//-----------------------------------------------------------------------------------------------------
//																
//									 	Tkmatik sp z o.o.
//
//	Name					:		FB_Save
//	Author					:		AM
//	Release Date			:		12.01.2022
//	Current ver				:		v 0.1
// 	Last correction 		:		12.01.2022
// 
//	Description				:
//		Special FB for saving structures to CSV files						
//
//	Requared hardware		:
//
// 	Configuration			:
//
//
//-----------------------------------------------------------------------------------------------------

FUNCTION_BLOCK FB_RecipeVariablesSaveCSV

VAR_INPUT
	bExecute							: BOOL := FALSE;(* Rising edge starts program execution *)
	sFilePath							: T_MaxString;(* CSV destination file path and name *)
//	database							: POINTER TO STRING(255);	
	nRows          						: UDINT;                // Liczba wierszy
    nCols          						: UDINT; 
	database							: POINTER TO STRING(255);//ARRAY[0..MAX_PARAMS_VARIABLES_COUNT-1] OF STRING(255);
	
END_VAR
VAR CONSTANT
	MAX_CSV_FIELD_LENGTH				: UDINT	:= 255;	
END_VAR
VAR_IN_OUT
END_VAR

VAR
	
	sNetId			: T_AmsNetId := '';	(* TwinCAT system network address *)
	sCSVLine		: T_MaxString := '';(* Single CSV text line (row, record), we are using string as record buffer (your are able to see created fields) *)
	sCSVField		: T_MaxString := '';(* Single CSV field value (column, record field) *)
	nRow	 		: UDINT 	:= 0;(* Row number (record) *)
	nColumn			: UDINT 	:= 0;(* Column number (record field) *)
	hFile			: UINT		:= 0;(* File handle of the source file *)
	step			: DWORD 	:= 0;
	fbFileOpen		: FB_FileOpen;(* Opens file *)
	fbFileClose		: FB_FileClose;(* Closes file *)
	fbFilePuts		: FB_FilePuts;(* Writes one record (line) *)
	fbWriter		: FB_CSVMemBufferWriter;(* Helper function block used to create CSV data bytes (single record line) *)
	rtExecute		:	R_TRIG;                         //	Rtrig for start



END_VAR
VAR_OUTPUT                                                                                  
	bBusy												:	BOOL;                           //	FB is Busy
	bDone												:	BOOL;                           //	Load cycle done, DATA actual 
	bError												:	BOOL;                           //	Flag error
	nErrId												:	UDINT;                          //	Error ID

END_VAR


rtExecute(CLK:=bExecute);
IF (NOT bExecute) THEN
	bDone												:=	FALSE;
END_IF

CASE step OF
	0:	(* Wait for rising edge at bWrite variable *)
		IF rtExecute.Q THEN
			bBusy 	:= TRUE;
			bError	:= FALSE;
			nErrId	:= 0;
			hFile	:= 0;
			nRow	:= 0;
			nColumn	:= 0;
			step 	:= 1;
		END_IF

	1:	(* Open source file *)
		fbFileOpen(  bExecute := FALSE  );
		fbFileOpen( sNetId := sNetId, sPathName := sFilePath, nMode := FOPEN_MODEWRITE OR FOPEN_MODETEXT,(* Open file in TEXT mode! *)
					ePath := PATH_GENERIC, bExecute := TRUE );
		step := 2;

	2:(* Wait until open not busy *)
		fbFileOpen( bExecute := FALSE, bError => bError, nErrID => nErrID, hFile => hFile );
		IF NOT fbFileOpen.bBusy THEN
			IF NOT fbFileOpen.bError THEN
				step := 3;
			ELSE(* Error: file not found? *)
				step := 100;
			END_IF
		END_IF

	3:(* Convert one PLC record to CSV format *)
		sCSVLine := '';
		fbWriter.eCmd := eEnumCmd_First;(* Write first field value *)
		IF nRow <= nRows THEN

			FOR nColumn := 0 TO nCols BY 1 DO
 
				sCSVField := STRING_TO_CSVFIELD( database[ nRow ], FALSE );(* TODO: Get field value from your application *)

				(* Add new field to the record buffer *)
				fbWriter( 	pBuffer := ADR( sCSVLine ), cbBuffer := SIZEOF( sCSVLine ) - 1, putValue := sCSVField, pValue := 0, cbValue := 0,
							bCRLF := ( nColumn = nCols ) );(* bCRLF == TRUE => Write CRLF after the last field value *)
				IF fbWriter.bOk THEN
					fbWriter.eCmd := eEnumCmd_Next;(* Write next field value *)
				ELSE(* Error *)
					step := 100;
					RETURN;
				END_IF

			END_FOR(* FOR nColumn := 0... *)

			(* FB_FilePuts adds allready CR (carriage return) to the written line.
			We have to replace the $R$L characters with $L character to avoid double CR. *)
			IF RIGHT( sCSVLine, 2 ) = '$R$L' THEN
				sCSVLine := REPLACE( sCSVLine, '$L', 2, LEN( sCSVLine ) - 1 );
			END_IF

			nRow := nRow + 1;(* Increment number of created records (rows) *)
			step := 4;(* Write record to the file *)

		ELSE(* All rows written => Close file *)
			step := 10;
		END_IF

	4:	(* Write single text line *)
		fbFilePuts( bExecute := FALSE );
		fbFilePuts( sNetId := sNetId, hFile := hFile, sLine := sCSVLine, bExecute := TRUE );
		step := 5;

	5:(* Wait until write not busy *)
		fbFilePuts( bExecute := FALSE, bError => bError, nErrID => nErrID );
		IF NOT fbFilePuts.bBusy THEN
			IF NOT fbFilePuts.bError THEN
				step := 3;(* Write next record *)
			ELSE(* Error *)
				step := 100;
			END_IF
		END_IF

	10:	(* Close source file *)
		fbFileClose( bExecute := FALSE );
		fbFileClose( sNetId := sNetId, hFile := hFile, bExecute := TRUE );
		step := 11;

	11:(* Wait until close not busy *)
		fbFileClose( bExecute := FALSE, bError => bError, nErrID => nErrID );
		IF ( NOT fbFileClose.bBusy ) THEN
			bDone	:= TRUE;
			hFile := 0;
			step := 100;
		END_IF

	100: (* Error or ready step => cleanup *)
		IF ( hFile <> 0 ) THEN
			step := 10; (* Close the source file *)
		ELSE
			bBusy := FALSE;
			step := 0;	(* Ready *)
		END_IF

END_CASE

END_FUNCTION_BLOCK

(* stored: Version 1.1.0.1, ProductVersion 3.1.4026.13, FileIdentifier 164c6e2f468b5e728ce9646aa66a136467f2319f, FileSignature 77334017cdd51c695b97f9433be66b5477b1b0db4353a412fa261df4bb14a7adcb77887bb7993f42f1a804e39ed593ed0f5c8e84284f29d0558bf9e52c599777f220740149fc77e2007397a26754a98388612da6dab6a30e04e81488361f34f666339e204c86defb3ca5cee5c941e7a2a02d78f4118827d0665a2584f3cc43fa707246533d57b3354714a3500657ba825bf670c3941ea1c0e4dfa096e598991bc71dd1c6a22012cf480339cb9f9db8069b2660af5648d0712d63ab7f1ebdf79f684ed13319ded1811842582057b3786c93ea6498ea48f9aa7c298a4019752a253b170ccf8547aa17c54964fefd7314f28645ac196992903efcba178e05bab8d5
   POU FB_RecipeVariablesSaveCSV: Id {e51e8360-ff65-4a05-8b97-048f37776386}, SpecialFunc None *)
